Universal Robots PolyScope program: 20250523.urp

Program 20250523 (installation=20240827 directory=/programs/con createdIn=5.15.1 lastSavedIn=5.15.1 robotSerialNumber=20245500285)
Calibrated DH parameters: a=[0.000097, -0.210459, -0.026602, 0.000137, 0.000078, 0]; d=[0.162601, 254.180657, -54.076236, -199.970743, 0.099615, 0.099684]; alpha=[1.569796, -0.001455, 0.001957, 1.570525, -1.571561, 0]; deltaTheta=[0, -1.053331, 8.839472, -1.50296, 0.000002, 0]
InitVariablesNode
Robot Program (runOnlyOnce=false)
  MoveJ speed 60 deg/s, acceleration 80 deg/s^2 (useActiveTCP=true) feature=Base
    Waypoint goudo: motionParameters(jointSpeed=1.047198 jointAcceleration=1.396263 cartesianSpeed=0.25 cartesianAcceleration=1.2); TCP in base x=804.816 y=122.737 z=261.364 mm, rx=1.21 ry=1.2107 rz=1.2121 rad; joints [178.646, -48.519, 103.06, -234.54, -88.651, 180.01] deg; TCP offset x=-0.17 y=0 z=192.95 mm, rx=0 ry=0 rz=0 rad
    Popup Message (haltProgram=false message=tcp inputType=Text)
    Waypoint tcp: TCP in base x=804.828 y=122.701 z=254.327 mm, rx=1.21 ry=1.2106 rz=1.2122 rad; joints [178.642, -47.721, 103.048, -235.329, -88.649, 180.01] deg
    x := 0.004
    y := 0.004
    z := 0.0002
    n := 1
    Loop Counting (count=20) loopVariable(name=循环_1)
      a1 := pose_add(tcp,p[0,0,-z*n-0.004,0,0,0])
      MoveJ speed 60 deg/s, acceleration 80 deg/s^2 (useActiveTCP=true) feature=Base
        Popup Message (haltProgram=false message=111 inputType=Text)
        Waypoint Variable (Variable): variable(name=a1)
        SuppressedNode
          Popup Message (haltProgram=false message=nnn inputType=Text)
        n := n+1
        SuppressedNode
          Popup Message (haltProgram=false message=nnnn inputType=Text)
    Popup Message (haltProgram=false message=000000 inputType=Text)
    SuppressedNode
      a1 := pose_add(tcp,p[0,0,-z*n,0,0,0])
    SuppressedNode
      MoveJ speed 60 deg/s, acceleration 80 deg/s^2 (useActiveTCP=true) feature=Base
        Popup Message (haltProgram=false message=111 inputType=Text)
        Waypoint Variable (Variable): variable=a1
        Popup Message (haltProgram=false message=222 inputType=Text)
    SuppressedNode
      a1 := p[0,0,-z*1,0,0,0]
    SuppressedNode
      a2 := p[0,0,-z*2,0,0,0]
    SuppressedNode
      a3 := p[0,0,-z*3,0,0,0]
    var_1 := p[0,0,-z*1,0,0,0]
    var_2 := p[0,0,-z*2,0,0,0]
    var_3 := p[0,0,-z*3,0,0,0]
    var_4 := p[0,0,-z*4,0,0,0]
    var_5 := p[0,0,-z*5,0,0,0]
    var_6 := p[0,0,-z*6,0,0,0]
    var_7 := p[0,0,-z*7,0,0,0]
    var_8 := p[0,0,-z*8,0,0,0]
    var_9 := p[0,0,-z*9,0,0,0]
    var_10 := p[0,0,-z*10,0,0,0]
    var_11 := p[0,0,-z*15,0,0,0]
    var_12 := p[0,0,-z*20,0,0,0]
    var_13 := p[0,0,-z*25,0,0,0]
    var_14 := p[0,0,-z*30,0,0,0]
    var_15 := p[0,0,-z*35,0,0,0]
    var_16 := p[0,0,-z*40,0,0,0]
    var_17 := p[0,0,-z*45,0,0,0]
    var_18 := p[0,0,-z*50,0,0,0]
    var_19 := p[0,0,-z*55,0,0,0]
    var_20 := p[0,0,-z*50,0,0,0]
    var_21 := p[0,0,-z*51,0,0,0]
    var_22 := p[0,0,-z*52,0,0,0]
    var_23 := p[0,0,-z*53,0,0,0]
    var_24 := p[0,0,-z*54,0,0,0]
    var_25 := p[0,0,-z*55,0,0,0]
    SuppressedNode
      b1 := p[x,y,-z*1,0,0,0]
    SuppressedNode
      b2 := p[x,y,-z*2,0,0,0]
    SuppressedNode
      b3 := p[x,y,-z*3,0,0,0]
    SuppressedNode
      c1 := p[-x,y,-z*1,0,0,0]
    SuppressedNode
      c2 := p[-x,y,-z*2,0,0,0]
    SuppressedNode
      c3 := p[-x,y,-z*3,0,0,0]
    SuppressedNode
      d1 := p[-x,-y,-z*1,0,0,0]
    SuppressedNode
      d2 := p[-x,-y,-z*2,0,0,0]
    SuppressedNode
      d3 := p[-x,-y,-z*3,0,0,0]
    SuppressedNode
      e1 := p[x,-y,-z*1,0,0,0]
    SuppressedNode
      e2 := p[x,-y,-z*2,0,0,0]
    SuppressedNode
      e3 := p[x,-y,-z*3,0,0,0]
    SuppressedNode
      tcpa1 := pose_add(tcp, a1)
    SuppressedNode
      tcpa2 := pose_add(tcp, a2)
    SuppressedNode
      tcpa3 := pose_add(tcp, a3)
    SuppressedNode
      tcpb1 := pose_add(tcp, b1)
    SuppressedNode
      tcpb2 := pose_add(tcp, b2)
    SuppressedNode
      tcpb3 := pose_add(tcp, b3)
    SuppressedNode
      tcpc1 := pose_add(tcp, c1)
    SuppressedNode
      tcpc2 := pose_add(tcp, c2)
    SuppressedNode
      tcpc3 := pose_add(tcp, c3)
    SuppressedNode
      tcpd1 := pose_add(tcp, d1)
    SuppressedNode
      tcpd2 := pose_add(tcp, d2)
    SuppressedNode
      tcpd3 := pose_add(tcp, d3)
    SuppressedNode
      tcpe1 := pose_add(tcp, e1)
    SuppressedNode
      tcpe2 := pose_add(tcp, e2)
    SuppressedNode
      tcpe3 := pose_add(tcp, e3)
    SuppressedNode
      MoveJ speed 60 deg/s, acceleration 80 deg/s^2 (useActiveTCP=true) feature=Base
        Popup Message (haltProgram=false message=az1 inputType=Text)
        Waypoint Variable (Variable): variable(name=tcpa1)
        Popup Message (haltProgram=false message=az2 inputType=Text)
        Waypoint Variable (Variable): variable(name=tcpa2)
        Popup Message (haltProgram=false message=az3 inputType=Text)
        Waypoint Variable (Variable): variable(name=tcpa3)
        Popup Message (haltProgram=false message=guodu inputType=Text)
        Waypoint goudo: TCP in base x=804.816 y=122.737 z=261.364 mm, rx=1.21 ry=1.2107 rz=1.2121 rad; joints [178.646, -48.519, 103.06, -234.54, -88.651, 180.01] deg
        Popup Message (haltProgram=false message=bz1 inputType=Text)
        Waypoint Variable (Variable): variable(name=tcpb1)
        Popup Message (haltProgram=false message=bz2 inputType=Text)
        Waypoint Variable (Variable): variable(name=tcpb2)
        Popup Message (haltProgram=false message=bz3 inputType=Text)
        Waypoint Variable (Variable): variable(name=tcpb3)
        Popup Message (haltProgram=false message=guodu inputType=Text)
        Waypoint goudo: TCP in base x=804.816 y=122.737 z=261.364 mm, rx=1.21 ry=1.2107 rz=1.2121 rad; joints [178.646, -48.519, 103.06, -234.54, -88.651, 180.01] deg
        Popup Message (haltProgram=false message=cz1 inputType=Text)
        Waypoint Variable (Variable): variable(name=tcpc1)
        Popup Message (haltProgram=false message=cz2 inputType=Text)
        Waypoint Variable (Variable): variable(name=tcpc2)
        Popup Message (haltProgram=false message=cz3 inputType=Text)
        Waypoint Variable (Variable): variable(name=tcpc3)
        Popup Message (haltProgram=false message=guodu inputType=Text)
        Waypoint goudo: TCP in base x=804.816 y=122.737 z=261.364 mm, rx=1.21 ry=1.2107 rz=1.2121 rad; joints [178.646, -48.519, 103.06, -234.54, -88.651, 180.01] deg
        Popup Message (haltProgram=false message=dz1 inputType=Text)
        Waypoint Variable (Variable): variable(name=tcpd1)
        Popup Message (haltProgram=false message=dz2 inputType=Text)
        Waypoint Variable (Variable): variable(name=tcpd2)
        Popup Message (haltProgram=false message=dz3 inputType=Text)
        Waypoint Variable (Variable): variable(name=tcpd3)
        Popup Message (haltProgram=false message=guodu inputType=Text)
        Waypoint goudo: TCP in base x=804.816 y=122.737 z=261.364 mm, rx=1.21 ry=1.2107 rz=1.2121 rad; joints [178.646, -48.519, 103.06, -234.54, -88.651, 180.01] deg
        Popup Message (haltProgram=false message=ez1 inputType=Text)
        Waypoint Variable (Variable): variable(name=tcpe1)
        Popup Message (haltProgram=false message=ez2 inputType=Text)
        Waypoint Variable (Variable): variable(name=tcpe2)
        Popup Message (haltProgram=false message=ez3 inputType=Text)
        Waypoint Variable (Variable): variable(name=tcpe3)
        Popup Message (haltProgram=false message=guodu inputType=Text)
